# EPICS autosave request: apps/vmeCratesApp/Db/vmeCratePedestal.req
$(PREF)t_set_mbbi
$(PREF)man_set_mbbi
$(PREF)cpid_param_mbbi
$(PREF)cpid_loc_mbbi
$(PREF)cpid_man_mbbi
$(PREF)cpid_dsbl_mbbi
$(PREF)cpid_loc_mod
$(PREF)cpid_dsbl
$(PREF)cpid.MMOD
$(PREF)t_set
$(PREF)cpid.KP
$(PREF)cpid.KI
$(PREF)cpid.KD
